// TIA Portal V19 export
TYPE "LEXCHANGETRAY_typeConstraintRollerIoSignalControlNode"
// reset: Bool
// monitoring: LEXCHANGETRAY_typeConstraintRollerIoSignalContronNodeMonitoring
// stored: Access Published
   STRUCT
      reset : Bool;
      monitoring { S7_SetPoint := 'True'} : "LEXCHANGETRAY_typeConstraintRollerIoSignalContronNodeMonitoring";
   END_STRUCT;
END_TYPE
